(* CODESYS project Fanuc_RPi.project

Project tree, tasks and I/O mapping:
  Device : CODESYS Control for Raspberry Pi MC SL, 3S - Smart Software Solutions GmbH, version 3.5.16.0
    application Application
      libraries: Standard, * (System); BASIC, 3.3.3.0 (OSCAT); MemoryUtils, 3.5.15.0 (3S - Smart Software Solutions GmbH); CoDeSys EIP, * (NothinRandom)
      task MainTask (cyclic, interval t#1ms, priority 1) calls PLC_PRG
      program PLC_PRG [ST]
      data type stStringRegister
      data type stJointPosition
      data type stCartesianPosition
      data type stAllRegistersINT
      data type stBlockRegistersINT
    SoftMotion General Axis Pool
    I²C
    SPI
    <Empty>
    Onewire
    Camera device
      <Empty>
  text list GlobalTextList
*)

// Device/Application/stStringRegister
{attribute 'pack_mode' := '4'}

// String struct
TYPE stStringRegister :
	STRUCT
		Length	: DINT;
		Data	: STRING;
	END_STRUCT
END_TYPE

// Device/Application/stJointPosition
{attribute 'pack_mode' := '0'}

// body		: 40B
// total	: 44B
// Joint position struct
TYPE stJointPosition :
	STRUCT
		UserFrame	: BYTE := 16#3F;
		ToolFrame	: BYTE := 16#1F;
		Reserved	: INT;
		J1			: REAL;
		J2			: REAL;
		J3			: REAL;
		J4			: REAL;
		J5			: REAL;
		J6			: REAL;
		// extended axis
		J7			: REAL;
		J8			: REAL;
		J9			: REAL;
	END_STRUCT
END_TYPE

// Device/Application/stCartesianPosition
{attribute 'pack_mode' := '0'}

// body		: 44B
// total	: 44B
// Cartesian position struct
TYPE stCartesianPosition :
	STRUCT
		UserFrame	: BYTE := 16#3F;
		ToolFrame	: BYTE := 16#1F;;
		Reserved	: INT;
		X			: REAL;
		Y			: REAL;
		Z			: REAL;
		Wx			: REAL;
		Py			: REAL;
		Rz			: REAL;
		TURN4		: SINT;
		TURN5		: SINT;
		TURN6		: SINT;
		// configuration
		RESERVED1 	: BIT;
		RESERVED2 	: BIT;
		RESERVED3 	: BIT;
		RESERVED4 	: BIT;
		FRONT	 	: BIT;
		UP		 	: BIT;
		LEFT	 	: BIT;
		FLIP	 	: BIT;
		// extended axis
		EXT1		: DINT;
		EXT2		: DINT;
		EXT3		: DINT;
	END_STRUCT
END_TYPE

// Device/Application/stAllRegistersINT
{attribute 'pack_mode' := '0'}

// body		: 496B
// total	: 496B
// numeric registers assuming type integer
TYPE stAllRegistersINT :
	STRUCT
		numRegs	: ARRAY [1..124] OF DINT;
	END_STRUCT
END_TYPE

// Device/Application/stBlockRegistersINT
{attribute 'pack_mode' := '0'}

// body		: 496B
// total	: 496B
// numeric registers assuming type integer
TYPE stBlockRegistersINT :
	STRUCT
		numRegs	: ARRAY [1..10] OF DINT;
	END_STRUCT
END_TYPE

// Device/Application/PLC_PRG
PROGRAM PLC_PRG
VAR
	_Robot 				: CoDeSys_EIP.Device(sIpAddress:='11.200.0.11', uiPort:=44818);
	_bEnable			: BOOL;					// enable function block
	_bAutoReconnect		: BOOL;					// enable auto session reconnect in case of timeout
	_bCloseSession		: BOOL;					// forward close and unregister session
	_bInit				: BOOL;					// one shot init
	_uiIndex			: UINT;					// state machine
	_bReadFinished		: BOOL;					// read status state
	_bWriteFinished		: BOOL;					// write status state
	_bGoodRead			: BOOL;					// status of read tag
	_bGoodWrite			: BOOL;					// status of write tag
	
	_sError				: STRING;				// function block's error message
	_bAckError			: BOOL;					// acknowledge error
	
	_stCipService		: CoDeSys_EIP.stCipService;
	_rNumReg			: REAL;					// test numeric register
	_diNumReg			: DINT;					// test numeric register
	_stStringRegister	: stStringRegister;		// test string register
	_stLPOS				: stCartesianPosition;	// current linear position
	_stJPOS				: stJointPosition;		// current joint position
	_stPosReg1			: stCartesianPosition;	// position register
	_stPosReg2			: stJointPosition;		// position register
	
	_stAllRegsInt		: stAllRegistersINT;	// contains 124 registers
	_stBlockRegsInt		: stBlockRegistersINT;	// contains 10 registers
END_VAR

(*

=====================
Service Code:
=====================
* 0x01 (1)	: get attribute all
* 0x02 (2)	: Set attribute all
* 0x0E (14)	: get attribute single
* 0x10 (16)	: set attribute single
* 0x32 (50)	: get attribute block
* 0x33 (51)	: set attribute block
=====================
Class Code:
=====================
* 0x6B (107) : numeric register integer
* 0x6C (108) : numeric register real
* 0x6D (109) : string register
* 0x7B (123) : position register (Cartesian)
* 0x7C (124) : position register (joint)
* 0x7D (125) : current position (Cartesian)
* 0x7E (126) : current position (joint)
=====================
Instance:
=====================
* 0x01 (1)		: single item
* 0x(len)(grp)	: block items (e.g. 0x0501 (1281) is for writing 5 items of group 1)
=====================
Attribute:
=====================
* 0x01 (1) 		: index of single item (if block items, then this is starting index)

*)

IF (NOT _bInit) THEN
	_bInit := TRUE;
	_Robot.bUnconnectedMessaging := TRUE; // only use Send RR Data!
END_IF

_Robot.bEnable := _bEnable;
_Robot.bAutoReconnect := _bAutoReconnect;

// perform forward close and unregister session
IF _bCloseSession THEN
	_bCloseSession := FALSE;
	_Robot.bCloseSession();
END_IF

_sError := _Robot.sError;
// acknowledge fault
IF _bAckError THEN
	_bAckError := FALSE;
	_Robot.bResetFault();
END_IF

_Robot(); // update _Robot.bEipCipActive

// all reads in one cycle
IF _Robot.bEipCipActive THEN
	WHILE (NOT _bReadFinished) DO
		// prevent stuck loop
		IF ((NOT _Robot.bEipCipActive) OR _Robot.bError) THEN
			EXIT;
		END_IF
		// read one tag at a time
		_bGoodRead := FALSE;
		// NOTE:
		//	* For numeric registers, you need to pick the data type
		//		* 0x6B (107) : numeric register integer
		//		* 0x6C (108) : numeric register real
		CASE _uiIndex OF
			0: // Read numeric register 5, which is an integer
				_stCipService.cipClass := 16#6B;
				_stCipService.instance := 16#01;
				_stCipService.attribute := 16#05; // register index 5
				_bGoodRead := _Robot.bGetAttributeSingle(stCipService:=_stCipService,
														pbBuffer:=ADR(_diNumReg),
														uiSize:=SIZEOF(_diNumReg),
														psId:=ADR('Read R#5: '));
			1: // Read numeric register 10, which is a real
				_stCipService.cipClass := 16#6C;
				_stCipService.instance := 16#01;
				_stCipService.attribute := 16#0A; // register index 10
				_bGoodRead := _Robot.bGetAttributeSingle(stCipService:=_stCipService,
															pbBuffer:=ADR(_rNumReg),
															uiSize:=SIZEOF(_rNumReg),
															psId:=ADR('Read R#10: '));
			2: // Read string register 5
				_stCipService.cipClass := 16#6D;
				_stCipService.instance := 16#01;
				_stCipService.attribute := 16#05; // register index 5
				_bGoodRead := _Robot.bGetAttributeSingle(stCipService:=_stCipService,
															pbBuffer:=ADR(_stStringRegister),
															uiSize:=SIZEOF(_stStringRegister),
															psId:=ADR('Read SR#5: '));
			3: // read position register 1 as cartesian position
				_stCipService.cipClass := 16#7B;
				_stCipService.instance := 16#01;
				_stCipService.attribute := 16#01; // register index 1
				_bGoodRead := _Robot.bGetAttributeSingle(stCipService:=_stCipService,
															pbBuffer:=ADR(_stPosReg1),
															uiSize:=SIZEOF(_stPosReg1),
															psId:=ADR('Read PR#1: '));
			4: // read position register 2 as joint position
				_stCipService.cipClass := 16#7C;
				_stCipService.instance := 16#01;
				_stCipService.attribute := 16#02; // register index 2
				_bGoodRead := _Robot.bGetAttributeSingle(stCipService:=_stCipService,
															pbBuffer:=ADR(_stPosReg2),
															uiSize:=SIZEOF(_stPosReg2),
															psId:=ADR('Read PR#2: '));
			5: // read current Cartesian position (LPOS)
				_stCipService.cipClass := 16#7D;
				_stCipService.instance := 16#01;
				_stCipService.attribute := 16#01;
				_bGoodRead := _Robot.bGetAttributeSingle(stCipService:=_stCipService,
															pbBuffer:=ADR(_stLPOS),
															uiSize:=SIZEOF(_stLPOS),
															psId:=ADR('Read LPOS: '));
			6: // read current joint position (JPOS)
				_stCipService.cipClass := 16#7E;
				_stCipService.instance := 16#01;
				_stCipService.attribute := 16#01;
				_bGoodRead := _Robot.bGetAttributeSingle(stCipService:=_stCipService,
															pbBuffer:=ADR(_stJPOS),
															uiSize:=SIZEOF(_stJPOS),
															psId:=ADR('Read JPOS: '));
			7: // read up to the first 124 registers
				_stCipService.cipClass := 16#6B; // change to 16#6C if you want to read as REAL
				_stCipService.instance := 16#01; // starting index of numeric register 1
				//_stCipService.attribute := 16#00; // optinal since method auto set to 0
				_bGoodRead := _Robot.bGetAttributeAll(stCipService:=_stCipService,
														pbBuffer:=ADR(_stAllRegsInt),
														uiSize:=SIZEOF(_stAllRegsInt),
														psId:=ADR('Read All INT: '));
			8: // read 10 numeric registers as integer starting from #101
				_stCipService.cipService := 16#32; // get attribute block
				_stCipService.cipClass := 16#6B; // numeric register (integer), change to 16#6C for real
				_stCipService.instance := 16#0A01; // 10 (16#0A) registers of group 1 (16#01)
				_stCipService.attribute := 16#65; // starting index 101
				_bGoodRead := _Robot.bGenericService(stCipService:=_stCipService,
														pbOutBuffer:=ADR(_stBlockRegsInt),
														uiOutSize:=SIZEOF(_stBlockRegsInt),
														psId:=ADR('Read 10 INT: '));
		ELSE
				_bReadFinished := TRUE;
				_uiIndex := 0;
		END_CASE
		// increment counter on successful read
		IF (_bGoodRead) THEN
			_uiIndex := _uiIndex + 1;
		END_IF
	END_WHILE
	// _bDataRead := FALSE; // optional
END_IF

// all writes in one cycle
IF _Robot.bEipCipActive THEN
	WHILE (NOT _bWriteFinished) DO
		// prevent stuck loop
		IF ((NOT _Robot.bEipCipActive) OR _Robot.bError) THEN
			EXIT;
		END_IF
		// write one tag at a time
		_bGoodWrite := FALSE;
		// NOTE:
		//	* For numeric registers, you need to pick the data type
		//		* 0x6B (107) : numeric register integer
		//		* 0x6C (108) : numeric register real
		CASE _uiIndex OF
			0: // write numeric register 5, which is an integer
				_stCipService.cipClass := 16#6B;
				_stCipService.instance := 16#01;
				_stCipService.attribute := 16#05; // register index 5
				_bGoodWrite := _Robot.bSetAttributeSingle(stCipService:=_stCipService,
															pbBuffer:=ADR(_diNumReg),
															uiSize:=SIZEOF(_diNumReg),
															psId:=ADR('Write R#5: '));
			1: // write numeric register 10, which is a real
				_stCipService.cipClass := 16#6C;
				_stCipService.instance := 16#01;
				_stCipService.attribute := 16#0A; // register index 10
				_bGoodWrite := _Robot.bSetAttributeSingle(stCipService:=_stCipService,
															pbBuffer:=ADR(_rNumReg),
															uiSize:=SIZEOF(_rNumReg),
															psId:=ADR('Write R#10: '));
			2: // write string register 5
				_stCipService.cipClass := 16#6D;
				_stCipService.instance := 16#01;
				_stCipService.attribute := 16#05; // register index 5
				_bGoodWrite := _Robot.bSetAttributeSingle(stCipService:=_stCipService,
															pbBuffer:=ADR(_stStringRegister),
															uiSize:=SIZEOF(_stStringRegister),
															psId:=ADR('Write SR#5: '));
			3: // write position register 1 as cartesian position
				_stCipService.cipClass := 16#7B;
				_stCipService.instance := 16#01;
				_stCipService.attribute := 16#01; // register index 1
				_bGoodWrite := _Robot.bSetAttributeSingle(stCipService:=_stCipService,
															pbBuffer:=ADR(_stPosReg1),
															uiSize:=SIZEOF(_stPosReg1),
															psId:=ADR('Write PR#1: '));
			4: // write position register 2 as joint position
				_stCipService.cipClass := 16#7C;
				_stCipService.instance := 16#01;
				_stCipService.attribute := 16#02; // register index 2
				_bGoodWrite := _Robot.bSetAttributeSingle(stCipService:=_stCipService,
															pbBuffer:=ADR(_stPosReg2),
															uiSize:=SIZEOF(_stPosReg2),
															psId:=ADR('Write PR#2: '));
			5: // write 10 numeric registers as integer starting from #101
				_stCipService.cipService := 16#33; // set attribute block
				_stCipService.cipClass := 16#6B; // numeric register (integer), change to 16#6C for real
				_stCipService.instance := 16#0A01; // 10 (16#0A) registers of group 1 (16#01)
				_stCipService.attribute := 16#65; // starting index 101
				_bGoodWrite := _Robot.bGenericService(stCipService:=_stCipService,
														pbInBuffer:=ADR(_stBlockRegsInt),
														uiInSize:=SIZEOF(_stBlockRegsInt),
														psId:=ADR('Write 10 INT: '));
		ELSE
				_bWriteFinished := TRUE;
				_uiIndex := 0;
		END_CASE
		// increment counter on successful write
		IF (_bGoodWrite) THEN
			_uiIndex := _uiIndex + 1;
		END_IF
	END_WHILE
	// _bDataWrite := FALSE; // optional
END_IF

END_PROGRAM
